SUBAPPLICATION Uebung_001g_AX (* DigitalInput_I1 negiert mit INIT und Delay auf DigitalOutput_Q1 *)
  (* Standard: 61499-2; Description: Copyright (c) 2023 Meisterschulen am Ostbahnhof This program and the accompanying materials are made available under the terms of the Eclipse Public License 2.0 which is available at https://www.eclipse.org/legal/epl-2.0/ SPDX-License-Identifier: EPL-2.0 *)
  (* Version 1.0, 2023-10-23, Franz Höpfinger, Meisterschulen am Ostbahnhof, initial API and implementation and/or initial documentation *)
  PACKAGE Uebungen;
  IMPORT logiBUS::io::DI::logiBUS_DI::Input_I1;
  IMPORT logiBUS::io::DQ::logiBUS_DO::Output_Q1;
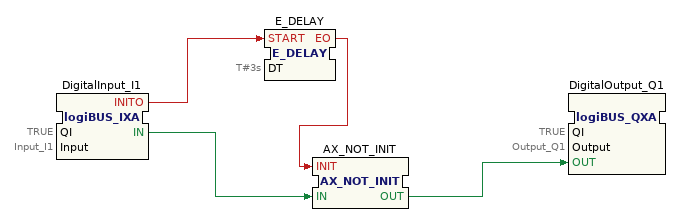
  (* obwohl I1 nicht abgefragt wird beim BOOT, wird AX_NOT hier TRUE ausgeben. *)
  FBS
    DigitalOutput_Q1 : logiBUS::io::DQ::logiBUS_QXA(QI := TRUE, Output := Output_Q1);
    DigitalInput_I1 : logiBUS::io::DI::logiBUS_IXA(QI := TRUE, Input := Input_I1);
    AX_NOT_INIT : adapter::booleanOperators::AX_NOT_INIT;
    E_DELAY : iec61499::events::E_DELAY(DT := T#3s);
  END_FBS
  EVENT_CONNECTIONS
    DigitalInput_I1.INITO TO E_DELAY.START;
    E_DELAY.EO TO AX_NOT_INIT.INIT;
  END_CONNECTIONS
  ADAPTER_CONNECTIONS
    DigitalInput_I1.IN TO AX_NOT_INIT.IN;
    AX_NOT_INIT.OUT TO DigitalOutput_Q1.OUT;
  END_CONNECTIONS
END_SUBAPPLICATION
